(* IEC 61131-3 sources: repolevel_ST_code_completion/output/20260127_205354/repoeval_traffic_light/readful_result, 3 files *)

(* ---- F_SecondsToTime.st ---- *)
FUNCTION F_SecondsToTime : TIME
VAR_INPUT
	dwSeconds	:	DWORD;		//输入的秒数
END_VAR
F_SecondsToTime := DWORD_TO_TIME(dwSeconds * 1000);
RETURN;
END_FUNCTION

(* ---- F_TimeToSeconds.st ---- *)
FUNCTION F_TimeToSeconds : DWORD
VAR_INPUT
	tTime	:	TIME;		//输入的时间
END_VAR
F_TimeToSeconds := DINT_TO_DWORD(TRUNC(TIME_TO_DWORD(tTime) / 1000.0));
RETURN;
END_FUNCTION

(* ---- FB_CountdownTimer.st ---- *)
FUNCTION_BLOCK FB_CountdownTimer
VAR_INPUT
	tElapsedTime	:	TIME;		//已经过的时间（定时器的ET）
	tTotalTime		:	TIME;		//总时间（定时器的PT）
END_VAR
VAR_OUTPUT
	nRemainingSeconds	:	UINT;	//剩余秒数
END_VAR
VAR
	nTotalSeconds		:	UINT;	//总秒数
	nElapsedSeconds		:	UINT;	//已过秒数
END_VAR

nTotalSeconds := INT_TO_UINT(TRUNC_INT(TIME_TO_DWORD(tTotalTime) / 1000.0));
nElapsedSeconds := INT_TO_UINT(TRUNC_INT(TIME_TO_DWORD(tElapsedTime) / 1000.0));

nRemainingSeconds := nTotalSeconds - nElapsedSeconds;
END_FUNCTION_BLOCK
